FUNCTION_BLOCK TableSerializerTest EXTENDS TcUnit.FB_TestSuite
VAR
END_VAR

SerializeTable();
SerializePartOfTableAndSwapColumnsAndWithoutHeader();

METHOD SerializePartOfTableAndSwapColumnsAndWithoutHeader : BOOL
VAR
	table : ARRAY[0..9] OF TestTableRow;
	i : INT;
	
	buffer : STRING(1000);
	sb : StringBuilderExtBuffer := (Buffer := ToAnyType(buffer));
	serializer : TableSerializer := (
		StringBuilder := sb
	);
	
	expected : STRING(1000);
END_VAR
TcUnit.TEST('Serialize part of table and swap columns');

// Prepare data
FOR i := 0 TO 9 DO
	table[i].timestamp := TO_TIME(i);
	table[i].value1 := i;
	table[i].value2 := i * 3.14;
	table[i].description := 'some text';
END_FOR

// Setup serialization
serializer.DecimalSeparator := ',';
serializer.Separator := ';';

// Bind data
serializer.DefineRow(table[0]);
serializer.RowCount := 7;
// Column order is different than structure
serializer.DefineNextColumn(table[0].description);
serializer.DefineNextColumn(table[0].timestamp);
serializer.DefineNextColumn(table[0].value2);

// Serialize
serializer.Serialize(includeHeader := FALSE, clearBuffer := TRUE);

expected := 'some text;T#0ms;0,0$Nsome text;T#1ms;3,14$Nsome text;T#2ms;6,28$Nsome text;T#3ms;9,42$Nsome text;T#4ms;12,56$Nsome text;T#5ms;15,700001$Nsome text;T#6ms;18,84';

AssertEquals_BOOL(
	Expected := TRUE,
	Actual := expected = buffer,
	Message := 'Table was not properly serialized');

TEST_FINISHED();
END_METHOD

METHOD SerializeTable : BOOL
VAR
	table : ARRAY[0..9] OF TestTableRow;
	i : INT;
	
	buffer : STRING(1000);
	sb : StringBuilderExtBuffer := (Buffer := ToAnyType(buffer));
	serializer : TableSerializer := (
		StringBuilder := sb
	);
	
	expected : STRING(1000);
END_VAR
TcUnit.TEST('Serialize table');

// Prepare data
FOR i := 0 TO 9 DO
	table[i].timestamp := TO_TIME(i);
	table[i].value1 := i;
	table[i].value2 := i * 3.14;
	table[i].description := 'some text';
END_FOR

// Setup serialization
serializer.DecimalSeparator := ',';
serializer.Separator := ';';

// Bind data
serializer.DefineRow(table[0]);
serializer.RowCount := 10;
serializer.DefineNextColumnWithName(table[0].timestamp, 'Timestamp');
serializer.DefineNextColumnWithName(table[0].value1, 'Value 1');
serializer.DefineNextColumnWithName(table[0].value2, 'Value 2');
serializer.DefineNextColumnWithName(table[0].description, 'Description');

// Serialize
serializer.Serialize(includeHeader := TRUE, clearBuffer := TRUE);

expected := 'Timestamp;Value 1;Value 2;Description$NT#0ms;0;0,0;some text$NT#1ms;1;3,14;some text$NT#2ms;2;6,28;some text$NT#3ms;3;9,42;some text$NT#4ms;4;12,56;some text$NT#5ms;5;15,700001;some text$NT#6ms;6;18,84;some text$NT#7ms;7;21,98;some text$NT#8ms;8;25,12;some text$NT#9ms;9;28,26;some text';

AssertEquals_BOOL(
	Expected := TRUE,
	Actual := expected = buffer,
	Message := 'Table was not properly serialized');

TEST_FINISHED();
END_METHOD

END_FUNCTION_BLOCK

(* stored: Version 1.1.0.1, ProductVersion 3.1.4024.15
   POU TableSerializerTest: Id {60732d81-9832-0c0c-031c-9a6aab1f515e}, SpecialFunc None
   Method SerializePartOfTableAndSwapColumnsAndWithoutHeader: Id {601e3b07-8459-01a5-069b-6d6bb0629397}
   Method SerializeTable: Id {b62053ff-5e49-0fbf-2b69-db083073aa3f} *)
